// TwinCAT 3 PLC project PLC
// ProgramVersion: 3.1.4023.0
// libraries:
//   Tc3_Module, * (Beckhoff Automation GmbH)
// project tree:
//   / Foo.TcPOU, PlcTask.TcTTO, Runner2.TcPOU, Runner1.TcPOU, Runner3.TcPOU, UsesFoo2.TcPOU, UsesFoo1.TcPOU, UsesFoo3.TcPOU
// real-time tasks:
//   TASK PlcTask: cycle T#10ms, priority 20, ADS port 350

CONFIGURATION PLC
    RESOURCE PLC ON TwinCAT3
        TASK PlcTask(INTERVAL := T#10ms, PRIORITY := 20);
        PROGRAM Runner2 WITH PlcTask : Runner2;
        PROGRAM Runner1 WITH PlcTask : Runner1;
        PROGRAM Runner3 WITH PlcTask : Runner3;
    END_RESOURCE
END_CONFIGURATION

// ---- Runner2.TcPOU
PROGRAM Runner2
VAR
    foo : Foo;
    usesFoo : UsesFoo2;
END_VAR

usesFoo(foo:=foo);

END_PROGRAM

// ---- Foo.TcPOU
FUNCTION_BLOCK Foo
VAR
    Counter : UINT := 0;
END_VAR

Counter := Counter + 1;

END_FUNCTION_BLOCK

// ---- UsesFoo2.TcPOU
FUNCTION_BLOCK UsesFoo2
VAR_IN_OUT
    foo : Foo;
END_VAR

foo();

END_FUNCTION_BLOCK

// ---- Runner1.TcPOU
PROGRAM Runner1
VAR
    usesFoo : UsesFoo1;
END_VAR

usesFoo();

END_PROGRAM

// ---- UsesFoo1.TcPOU
FUNCTION_BLOCK UsesFoo1
VAR_INPUT
    foo : REFERENCE TO Foo;
END_VAR

IF __ISVALIDREF(foo) THEN
    foo();
END_IF

END_FUNCTION_BLOCK

// ---- Runner3.TcPOU
PROGRAM Runner3
VAR
    foo : Foo;
    usesFoo : UsesFoo3(foo);
END_VAR

usesFoo();

END_PROGRAM

// ---- UsesFoo3.TcPOU
FUNCTION_BLOCK UsesFoo3
VAR
    _foo : REFERENCE TO Foo;
END_VAR

_foo();

METHOD FB_init : BOOL
VAR_INPUT
	bInitRetains : BOOL; // if TRUE, the retain variables are initialized (warm start / cold start)
	bInCopyCode : BOOL;  // if TRUE, the instance afterwards gets moved into the copy code (online change)
    foo : REFERENCE TO Foo;
END_VAR
_foo REF= foo;
END_METHOD

END_FUNCTION_BLOCK
